// TIA Portal project "Lepteto motor teljes" (V15.1)

(* hardware
DEVICE "HMI_1"  KTP600 Basic color PN
   slot 0: "HMI_1"  KTP600 Basic color PN  6AV6 647-0AD11-3AX0  12.0.0.0
   slot 1: "HMI_RT_1"  KTP600 Basic color PN  6AV6 647-0AD11-3AX0  12.0.0.0
   slot 5: "HMI_1.IE_CP_1"  PROFINET Interface  12.0.0.0
      slot 1: "PROFINET Interface_1"  PROFINET Interface
         slot 1: "Port_1"  Port
DEVICE "S7300/ET200M station_2"  S7-300 station
   slot 0: "Rail_0"  Rail  6ES7 390-1***0-0AA0
   slot 2: "PLC_2"  CPU 314C-2 PN/DP  6ES7 314-6EH04-0AB0  V3.3
      slot 2: "PROFINET interface_1"  PN-IO
         slot 1: "Port_1"  Port
         slot 2: "Port_2"  Port
      slot 5: "DI 24/DO 16_1"  DI24/DO16
      slot 6: "AI 5/AO 2_1"  AI5/AO2
      slot 7: "Count_1"  Counter
      slot 8: "Positioning_1"  Positioning
*)

// ===== PLC "PLC_2"  CPU 314C-2 PN/DP =====

VAR_GLOBAL   // PLC tag table "Default tag table_1"
   "Orajel" AT %M0.5 : Bool;
   "Start" AT %M2.3 : Bool;
   "Kimenet" AT %Q136.0 : Bool;
   "Segedvaltozo" AT %M1.1 : Bool;
   "Eloirt" AT %MW37 : Int;
   "Aktualis" AT %MW4 : Int;
   "Ok" AT %M1.2 : Bool;
   "Felfele" AT %M1.3 : Bool;
   "Lefele" AT %M1.4 : Bool;
   "Sebesseg" AT %MW6 : Int;
   "Periodus" AT %MW8 : S5Time;
   "T1" AT %MW10 : S5Time;
   "T2" AT %MW12 : S5Time;
   "Vezerlo kimenet" AT %QW44 : Int;
END_VAR

VAR_GLOBAL   // PLC tag table "Default tag table"
   "Tag_1" AT %T1 : Timer;
   "Tag_2" AT %T2 : Timer;
   "Tag_3" AT %M10.0 : Bool;
   "Tag_4" AT %M10.1 : Bool;
   "Tag_5" AT %M14.1 : Bool;
   "Teszt1" AT %MW18 : Int;
   "Teszt2" AT %MW20 : Int;
   "Periodus1" AT %MD22 : Time;
   "Irany" AT %Q136.1 : Bool;
END_VAR

VAR_GLOBAL   // PLC tag table "Tag table_1"
   "Startbit" AT %M14.0 : Bool;
   "Start1" AT %M14.2 : Bool;
   "Start2" AT %M14.3 : Bool;
   "Start3" AT %M14.4 : Bool;
   "OK(1)" AT %M14.5 : Bool;
   "AlfaStart" AT %M14.6 : Bool;
   "Felfele2" AT %M14.7 : Bool;
END_VAR

ORGANIZATION_BLOCK "Main"   // OB1, LAD
TITLE = "Main Program Sweep (Cycle)"
{ S7_Optimized_Access := 'FALSE' }
VERSION : 0.1
   VAR_TEMP
      OB1_EV_CLASS : Byte;   // Bits 0-3 = 1 (Coming event), Bits 4-7 = 1 (Event class 1)
      OB1_SCAN_1 : Byte;   // 1 (Cold restart scan 1 of OB 1), 3 (Scan 2-n of OB 1)
      OB1_PRIORITY : Byte;   // Priority of OB Execution
      OB1_OB_NUMBR : Byte;   // 1 (Organization block 1, OB1)
      OB1_RESERVED_1 : Byte;   // Reserved for system
      OB1_RESERVED_2 : Byte;   // Reserved for system
      OB1_PREV_CYCLE : Int;   // Cycle time of previous OB1 scan (milliseconds)
      OB1_MIN_CYCLE : Int;   // Minimum cycle time of OB1 (milliseconds)
      OB1_MAX_CYCLE : Int;   // Maximum cycle time of OB1 (milliseconds)
      OB1_DATE_TIME : Date_And_Time;   // Date and time OB1 started
   END_VAR
   VAR_TEMP   // added for the SCL form of the ladder/FBD networks
      _w1 : Bool;
      _w2 : Bool;
      _w3 : Bool;
      _s5time1 : S5Time;
   END_VAR
BEGIN

REGION Network 1 (STL)
         L     "Sebesseg";
         ITB;
         L     W#16#0FFF;
         AW;
         L     W#16#1000;
         OW;
         T     "Periodus";
END_REGION

REGION Network 2
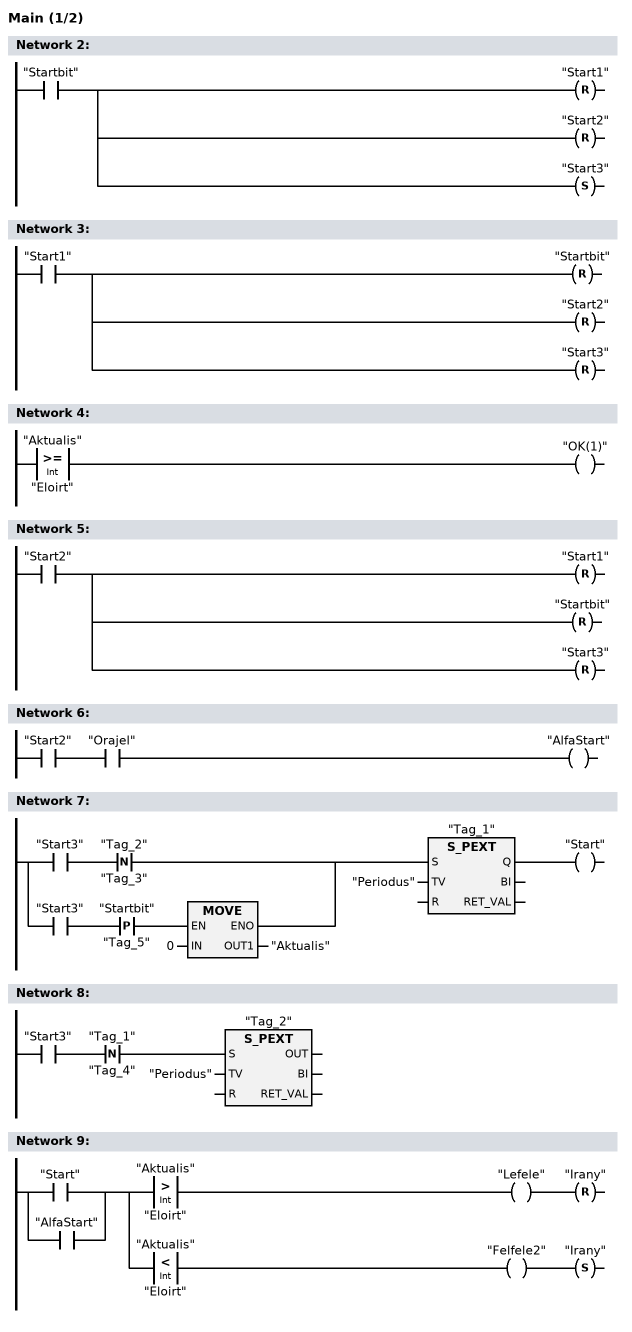
   RUNG wire#powerrail
      Contact( "Startbit" )
      wire#w1
      R_Coil( "Start1" )
   END_RUNG
   RUNG wire#w1
      R_Coil( "Start2" )
   END_RUNG
   RUNG wire#w1
      S_Coil( "Start3" )
   END_RUNG
   // the same network as SCL:
   IF "Startbit" THEN
       "Start1" := FALSE;
       "Start2" := FALSE;
       "Start3" := TRUE;
   END_IF;
END_REGION

REGION Network 3
   RUNG wire#powerrail
      Contact( "Start1" )
      wire#w1
      R_Coil( "Startbit" )
   END_RUNG
   RUNG wire#w1
      R_Coil( "Start2" )
   END_RUNG
   RUNG wire#w1
      R_Coil( "Start3" )
   END_RUNG
   // the same network as SCL:
   IF "Start1" THEN
       "Startbit" := FALSE;
       "Start2" := FALSE;
       "Start3" := FALSE;
   END_IF;
END_REGION

REGION Network 4
   RUNG wire#powerrail
      { S7_Templates := "SrcType := Int" } GE_Contact(in1 := "Aktualis", in2 := "Eloirt")
      Coil( "OK(1)" )
   END_RUNG
   // the same network as SCL:
   "OK(1)" := "Aktualis" >= "Eloirt";
END_REGION

REGION Network 5
   RUNG wire#powerrail
      Contact( "Start2" )
      wire#w1
      R_Coil( "Start1" )
   END_RUNG
   RUNG wire#w1
      R_Coil( "Startbit" )
   END_RUNG
   RUNG wire#w1
      R_Coil( "Start3" )
   END_RUNG
   // the same network as SCL:
   IF "Start2" THEN
       "Start1" := FALSE;
       "Startbit" := FALSE;
       "Start3" := FALSE;
   END_IF;
END_REGION

REGION Network 6
   RUNG wire#powerrail
      Contact( "Start2" )
      Contact( "Orajel" )
      Coil( "AlfaStart" )
   END_RUNG
   // the same network as SCL:
   "AlfaStart" := "Start2" AND "Orajel";
END_REGION

REGION Network 7
   RUNG wire#powerrail
      Contact( "Start3" )
      N_Contact(operand := "Tag_2", bit := "Tag_3")
      wire#w1
      S_PEXT(T_NO := "Tag_1", TV := "Periodus", R :=, BI =>, RET_VAL =>)
      Coil( "Start" )
   END_RUNG
   RUNG wire#powerrail
      Contact( "Start3" )
      P_Contact(operand := "Startbit", bit := "Tag_5")
      { S7_GenerateENO := "TRUE" } Move(in := 0, out1 => "Aktualis")
   END_RUNG wire#w1
   // the same network as SCL:
   // ENO of a box is taken as its EN; it also drops when the box reports an error
   #_w1 := "Start3" AND NOT "Tag_2" AND "Tag_3";   // falling edge of "Tag_2"
   "Tag_3" := "Tag_2";
   #_w2 := "Start3" AND "Startbit" AND NOT "Tag_5";   // rising edge of "Startbit"
   "Tag_5" := "Startbit";
   IF #_w2 THEN "Aktualis" := 0; END_IF;
   #_s5time1 := S_PEXT(T_NO := "Tag_1", S := #_w1 OR #_w2, TV := "Periodus", Q => #_w3);
   "Start" := #_w3;
END_REGION

REGION Network 8
   RUNG wire#powerrail
      Contact( "Start3" )
      N_Contact(operand := "Tag_1", bit := "Tag_4")
      S_PEXT(T_NO := "Tag_2", TV := "Periodus", R :=, BI =>, RET_VAL =>)
   END_RUNG
   // the same network as SCL:
   #_w1 := "Start3" AND NOT "Tag_1" AND "Tag_4";   // falling edge of "Tag_1"
   "Tag_4" := "Tag_1";
   #_s5time1 := S_PEXT(T_NO := "Tag_2", S := #_w1, TV := "Periodus");
END_REGION

REGION Network 9
   RUNG wire#powerrail
      Contact( "Start" )
      wire#w1
      { S7_Templates := "SrcType := Int" } GT_Contact(in1 := "Aktualis", in2 := "Eloirt")
      Coil( "Lefele" )
      R_Coil( "Irany" )
   END_RUNG
   RUNG wire#powerrail
      Contact( "AlfaStart" )
   END_RUNG wire#w1
   RUNG wire#w1
      { S7_Templates := "SrcType := Int" } LT_Contact(in1 := "Aktualis", in2 := "Eloirt")
      Coil( "Felfele2" )
      S_Coil( "Irany" )
   END_RUNG
   // the same network as SCL:
   #_w1 := "Start" OR "AlfaStart";
   "Lefele" := #_w1 AND ("Aktualis" > "Eloirt");
   IF "Lefele" THEN "Irany" := FALSE; END_IF;
   "Felfele2" := #_w1 AND ("Aktualis" < "Eloirt");
   IF "Felfele2" THEN "Irany" := TRUE; END_IF;
END_REGION

REGION Network 10
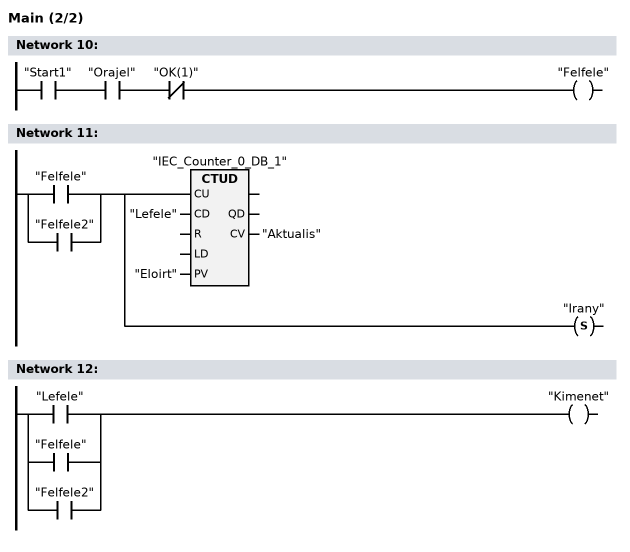
   RUNG wire#powerrail
      Contact( "Start1" )
      Contact( "Orajel" )
      I_Contact( "OK(1)" )
      Coil( "Felfele" )
   END_RUNG
   // the same network as SCL:
   "Felfele" := "Start1" AND "Orajel" AND NOT "OK(1)";
END_REGION

REGION Network 11
   #_w1 := "Felfele" OR "Felfele2";
   "IEC_Counter_0_DB_1".CTUD(CU := #_w1, CD := "Lefele", PV := "Eloirt", CV => "Aktualis");
   IF #_w1 THEN "Irany" := TRUE; END_IF;
END_REGION

REGION Network 12
   RUNG wire#powerrail
      Contact( "Lefele" )
      wire#w1
      Coil( "Kimenet" )
   END_RUNG
   RUNG wire#powerrail
      Contact( "Felfele" )
   END_RUNG wire#w1
   RUNG wire#powerrail
      Contact( "Felfele2" )
   END_RUNG wire#w1
   // the same network as SCL:
   "Kimenet" := "Lefele" OR "Felfele" OR "Felfele2";
END_REGION
END_ORGANIZATION_BLOCK

(* ===== HMI "HMI_RT_1" =====
system functions are stored by id; their names below are inferred from use
connection "HMI_Connection_1": ETHERNET, SIMATIC S7 300/400 MPI

HMI tags "Default tag table"
   "Eloirt" : Int = PLC Eloirt AT %MW37, 100 ms
   "Aktualis" : Int = PLC Aktualis AT %MW4, 100 ms
   "Sebesseg" : Int = PLC Sebesseg AT %MW6, 100 ms
   "Start1" : Bool = PLC Start1 AT %M14.2, 100 ms
   "Startbit" : Bool = PLC Startbit AT %M14.0, 100 ms
   "Start2" : Bool = PLC Start2 AT %M14.3, 100 ms
   "Kimenet" : Bool = PLC Kimenet AT %Q136.0, 100 ms
   "Irany" : Bool = PLC Irany AT %Q136.1, 100 ms
   "Start3" : Bool = PLC Start3 AT %M14.4, 100 ms

screen "Root screen" 320x240, template "Template_1"
   TextField "HmiScreenItemData" at 32,34 size 256x44; Text 'Léptető motor vezérlés'
   Button "Button_1" at 32,95 size 107x30; TextOff 'Csak előre'
      on Press: ActivateScreen("Screen_1", 0)
   Button "Button_2" at 188,95 size 107x30; TextOff 'Előre-hátra'
      on Press: ActivateScreen("Screen_2", 0)
   Button "Button_3" at 64,144 size 215x33; TextOff 'Előre Hátra változó frekvenciával'
      on Press: ActivateScreen("Screen_3", 0)

Template "Template_1" 320x240
   Button "Exit" at 266,202 size 52x37; TextOn 'Exit'; TextOff 'Exit'; PictureOn "ExitRuntime_KTP600_Basic_color_PN"; PictureOff "ExitRuntime_KTP600_Basic_color_PN"
      on Release: StopRuntime(0)
   Button "Template_Button" at 213,202 size 52x37; TextOff 'Text'
   Button "Template_Button_1" at 160,202 size 52x37; TextOff 'Text'
   Button "Template_Button_2" at 107,202 size 52x37; TextOff 'Text'
   Button "Start screen" at 54,202 size 52x37; TextOn 'Start screen'; TextOff 'Start screen'; PictureOn "NavigateHome_KTP600_Basic_color_PN"; PictureOff "NavigateHome_KTP600_Basic_color_PN"
      on Release: ActivateScreen("Root screen", 0)
   Button "Alarms" at 1,202 size 52x37; TextOn 'Alarms'; TextOff 'Alarms'; PictureOn "AlarmDisplay_KTP600_Basic_color_PN"; PictureOff "AlarmDisplay_KTP600_Basic_color_PN"
      on Release: function_ef3f5d25("Alarm window_Unacknowledged", -1)
   DateTimeField "HmiScreenItemData" at 235,19 size 85x19
   DateTimeField "HmiScreenItemData_1" at 235,0 size 85x19
   GraphicView "Logo" at 0,0 size 67x38; Picture "Logo of HMI_1"

screen "Screen_1" 320x240
   TextField "HmiScreenItemData" at 31,42 size 256x44; Text 'Léptető motor vezérlés'
   TextField "HmiScreenItemData_1" at 0,72 size 120x44; Text 'Előírt lépésszám:'
   TextField "HmiScreenItemData_2" at 8,108 size 120x44; Text 'Aktuális lépésszám:'
   IOField "I/O field_1" at 123,121 size 44x18; FormatPattern s99999
      ProcessValue <- "Aktualis"
   IOField "I/O field_2" at 117,82 size 96x23; FormatPattern s99999
      ProcessValue <- "Eloirt"
   Button "Button_1" at 104,158 size 96x32; TextOff 'Start'
      on Press: SetBit("Start1")
   Button "Button_2" at 114,198 size 76x25; TextOff 'Home'
      on Press: ActivateScreen("Root screen", 0); ResetBit("Start1"); ResetBit("Start2"); ResetBit("Startbit"); ResetBit("Start3")
   Circle "Circle_1" at 232,147 size 25x25
      Appearance <- "Kimenet"
   TextField "HmiScreenItemData_3" at 213,121 size 72x29; Text 'Kimenet'
   Circle "Circle_2" at 233,190 size 25x25
      Appearance <- "Irany"
   TextField "HmiScreenItemData_4" at 215,160 size 72x42; Text 'Irány'

screen "Screen_3" 320x240
   TextField "HmiScreenItemData" at 32,10 size 256x44; Text 'Léptető motor vezérlés'
   TextField "HmiScreenItemData_1" at 1,40 size 120x44; Text 'Előírt lépésszám:'
   TextField "HmiScreenItemData_2" at 9,67 size 120x44; Text 'Aktuális lépésszám:'
   IOField "I/O field_1" at 124,80 size 44x18; FormatPattern s99999
      ProcessValue <- "Aktualis"
   IOField "I/O field_2" at 118,50 size 96x23; FormatPattern s99999
      ProcessValue <- "Eloirt"
   TextField "HmiScreenItemData_3" at 9,92 size 120x44; Text 'Sebesseg:'
   IOField "I/O field_3" at 120,105 size 96x23; FormatPattern 99999
      ProcessValue <- "Sebesseg"
   Button "Button_1" at 116,149 size 96x32; TextOff 'Start'
      on Press: SetBit("Startbit")
   Circle "Circle_1" at 232,154 size 25x25
      Appearance <- "Kimenet"
   Circle "Circle_2" at 233,197 size 25x25
      Appearance <- "Irany"
   TextField "HmiScreenItemData_4" at 215,176 size 72x26; Text 'Irány'
   TextField "HmiScreenItemData_5" at 213,123 size 72x42; Text 'Kimenet'
   Button "Button_2" at 126,191 size 76x25; TextOff 'Home'
      on Press: ActivateScreen("Root screen", 0); ResetBit("Start1"); ResetBit("Start2"); ResetBit("Startbit"); ResetBit("Start3")
   TextField "HmiScreenItemData_6" at 190,92 size 120x44; Text '* 100 ms'

screen "Screen_2" 320x240
   TextField "HmiScreenItemData" at 31,42 size 256x44; Text 'Léptető motor vezérlés'
   TextField "HmiScreenItemData_1" at 0,72 size 120x44; Text 'Előírt lépésszám:'
   TextField "HmiScreenItemData_2" at 8,108 size 120x44; Text 'Aktuális lépésszám:'
   IOField "I/O field_1" at 123,121 size 44x18; FormatPattern s99999
      ProcessValue <- "Aktualis"
   IOField "I/O field_2" at 117,82 size 96x23; FormatPattern s99999
      ProcessValue <- "Eloirt"
   Button "Button_1" at 104,158 size 96x32; TextOff 'Start'
      on Press: SetBit("Start2"); ResetBit("Start1")
   Circle "Circle_1" at 232,147 size 25x25
      Appearance <- "Kimenet"
   Circle "Circle_2" at 233,190 size 25x25
      Appearance <- "Irany"
   TextField "HmiScreenItemData_4" at 215,160 size 72x42; Text 'Irány'
   TextField "HmiScreenItemData_3" at 213,124 size 72x26; Text 'Kimenet'
   Button "Button_2" at 114,198 size 76x25; TextOff 'Home'
      on Press: ActivateScreen("Root screen", 0); ResetBit("Start1"); ResetBit("Start2"); ResetBit("Startbit"); ResetBit("Start3")
*)